(* Schneider Machine Expert - Basic project FINAL_MIXER, file version 2.2.0.0 *)
(* ProjectInformations: Name=New project *)

HARDWARE
  Cpu 0: TM221CE40T
  EthernetConfiguration: NetworkName=M221, IpAllocationMode=FixedAddress, IpAddress=0.0.0.0, SubnetMask=0.0.0.0
  SerialLineConfiguration: Baud=Baud19200, Parity=ParityEven, DataBits=DataBits8, StopBits=StopBits1, PhysicalMedium=PhysicalMediumRs485, TransmissionMode=TransmissionModeModbusRtu, SlaveId=1, Addressing=SlaveAddressing
  MastTask: UsePeriodScanMode=false, PeriodScan=100
  FastTask: Period=255
  CpuBehavior: StartingMode=StartAsPreviousState, AutoSaveRamOnEeprom=true, WatchdogPeriod=250

SYMBOLS  (address, symbol, comment, settings)
  %M0       VACIAR_MEZCLA
  %M1       REINICIAR_CICLO
  %TM0      TM_INICIO_PROCESO  [Preset=3, Base=OneSecond]
  %TM1      TM_ESPERAR_VERTER  [Type=TP, Preset=5, Base=OneSecond]
  %TM2      TM_MEZCLANDO  [Type=TP, Preset=10, Base=OneSecond]
  %TM3      TM_ESPERAR_VACIAR  [Type=TOF, Preset=10, Base=OneSecond]
  %I0.0     BTN_INICIAR_PROCESO
  %I0.1     SENSOR_NIVEL_ALTO
  %I0.2     SENSOR_MAS_1
  %I0.3     SENSOR_MAS_2
  %I0.4     INICIAR_MIX
  %I0.5     DET_PROCESO
  %I0.8     SENSOR_TANQ_VACIO
  %Q0.0     LED_TRABAJANDO
  %Q0.1     LED_NIVEL_ALTO
  %Q0.2     LED_MEZCLANDO
  %Q0.4     VALV_PROD_A
  %Q0.5     VALV_PROD_B
  %Q0.6     MOT_1_COMP_BASC
  %Q0.7     MOT_2_MEZCLAR
  %Q0.8     VALV_ENTRADA_H2O
  %Q0.9     VALV_VACIAR_TANQ

POU New POU
  (* SectionNumber=1 *)

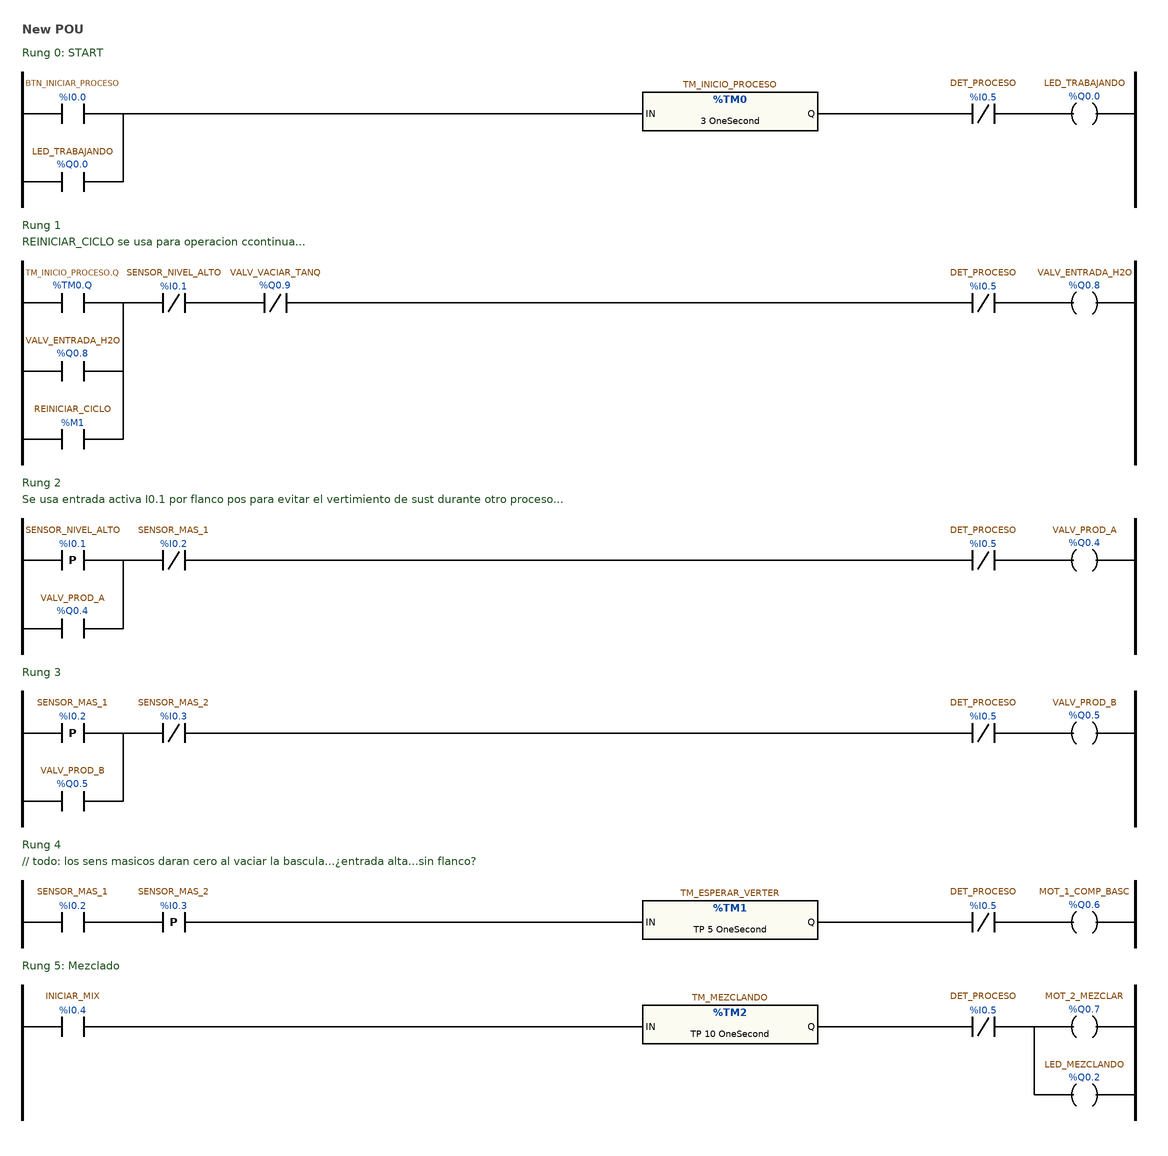

// Rung 0: START
  BLK %TM0                (* TM_INICIO_PROCESO *)
  LD %I0.0                (* BTN_INICIAR_PROCESO *)
  OR %Q0.0                (* LED_TRABAJANDO *)
  IN
  OUT_BLK
  LD Q
  ANDN %I0.5              (* DET_PROCESO *)
  ST %Q0.0                (* LED_TRABAJANDO *)
  END_BLK
  // as ST:
  //   TM_INICIO_PROCESO(IN := BTN_INICIAR_PROCESO OR LED_TRABAJANDO);
  //   LED_TRABAJANDO := TM_INICIO_PROCESO.Q AND NOT DET_PROCESO;

// Rung 1
// REINICIAR_CICLO se usa para operacion ccontinua...
  LD %TM0.Q               (* TM_INICIO_PROCESO *)
  OR %Q0.8                (* VALV_ENTRADA_H2O *)
  OR %M1                  (* REINICIAR_CICLO *)
  ANDN %I0.1              (* SENSOR_NIVEL_ALTO *)
  ANDN %Q0.9              (* VALV_VACIAR_TANQ *)
  ANDN %I0.5              (* DET_PROCESO *)
  ST %Q0.8                (* VALV_ENTRADA_H2O *)
  // as ST:
  //   VALV_ENTRADA_H2O := (TM_INICIO_PROCESO.Q OR VALV_ENTRADA_H2O OR REINICIAR_CICLO) AND NOT SENSOR_NIVEL_ALTO AND NOT VALV_VACIAR_TANQ AND NOT DET_PROCESO;

// Rung 2
// Se usa entrada activa I0.1 por flanco pos para evitar el vertimiento de sust durante otro proceso...
  LDR %I0.1               (* SENSOR_NIVEL_ALTO *)
  OR %Q0.4                (* VALV_PROD_A *)
  ANDN %I0.2              (* SENSOR_MAS_1 *)
  ANDN %I0.5              (* DET_PROCESO *)
  ST %Q0.4                (* VALV_PROD_A *)
  // as ST:
  //   VALV_PROD_A := (RISING(SENSOR_NIVEL_ALTO) OR VALV_PROD_A) AND NOT SENSOR_MAS_1 AND NOT DET_PROCESO;

// Rung 3
  LDR %I0.2               (* SENSOR_MAS_1 *)
  OR %Q0.5                (* VALV_PROD_B *)
  ANDN %I0.3              (* SENSOR_MAS_2 *)
  ANDN %I0.5              (* DET_PROCESO *)
  ST %Q0.5                (* VALV_PROD_B *)
  // as ST:
  //   VALV_PROD_B := (RISING(SENSOR_MAS_1) OR VALV_PROD_B) AND NOT SENSOR_MAS_2 AND NOT DET_PROCESO;

// Rung 4
// // todo: los sens masicos daran cero al vaciar la bascula...¿entrada alta...sin flanco?
  BLK %TM1                (* TM_ESPERAR_VERTER *)
  LD %I0.2                (* SENSOR_MAS_1 *)
  ANDR %I0.3              (* SENSOR_MAS_2 *)
  IN
  OUT_BLK
  LD Q
  ANDN %I0.5              (* DET_PROCESO *)
  ST %Q0.6                (* MOT_1_COMP_BASC *)
  END_BLK
  // as ST:
  //   TM_ESPERAR_VERTER(IN := SENSOR_MAS_1 AND RISING(SENSOR_MAS_2));
  //   MOT_1_COMP_BASC := TM_ESPERAR_VERTER.Q AND NOT DET_PROCESO;

// Rung 5: Mezclado
  BLK %TM2                (* TM_MEZCLANDO *)
  LD %I0.4                (* INICIAR_MIX *)
  IN
  OUT_BLK
  LD Q
  ANDN %I0.5              (* DET_PROCESO *)
  ST %Q0.7                (* MOT_2_MEZCLAR *)
  ST %Q0.2                (* LED_MEZCLANDO *)
  END_BLK
  // as ST:
  //   TM_MEZCLANDO(IN := INICIAR_MIX);
  //   MOT_2_MEZCLAR := TM_MEZCLANDO.Q AND NOT DET_PROCESO;
  //   LED_MEZCLANDO := TM_MEZCLANDO.Q AND NOT DET_PROCESO;

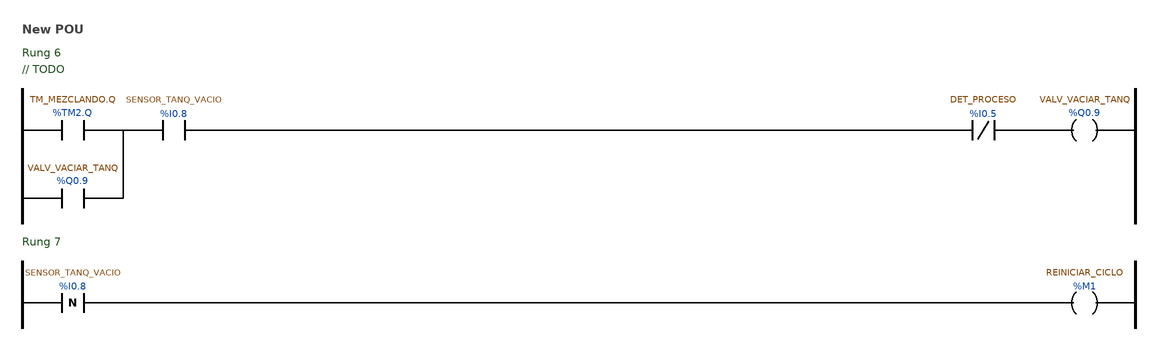

// Rung 6
// // TODO
  LD %TM2.Q               (* TM_MEZCLANDO *)
  OR %Q0.9                (* VALV_VACIAR_TANQ *)
  AND %I0.8               (* SENSOR_TANQ_VACIO *)
  ANDN %I0.5              (* DET_PROCESO *)
  ST %Q0.9                (* VALV_VACIAR_TANQ *)
  // as ST:
  //   VALV_VACIAR_TANQ := (TM_MEZCLANDO.Q OR VALV_VACIAR_TANQ) AND SENSOR_TANQ_VACIO AND NOT DET_PROCESO;

// Rung 7
  LDF %I0.8               (* SENSOR_TANQ_VACIO *)
  ST %M1                  (* REINICIAR_CICLO *)
  // as ST:
  //   REINICIAR_CICLO := FALLING(SENSOR_TANQ_VACIO);
